Staubli VAL3: page_inOut.dtx

bool bButton[8]
  [6] = true
  [7] = true
bool bLarge = true
num nIndex
num nInsert
num nKey = -1
public num nPage
num nRefresh
num nSelected = -1
num nTime = 0.5
num nView
num nViewMode = 1
string sEvent
public string sItems
string sList
string sMenu[8]
  [6] = "Delete"
  [7] = "New"
string sMenu8[8]
string sMessage
string sMode = "OUT"
string sId
